// TIA Portal V20 export
FUNCTION_BLOCK "LER_BrakeTest"   // FB103, LAD
// stored: Access Published, MemoryReserve 100, SetENOAutomatically false
   VAR_INPUT
      unitStatus : "LAF_typeUnitStatus";   // Status of the unit
      EnableManualCmds : Bool;
      mcRun : Bool;
      allFDoorClose : Bool;
      allFDoorRelease : Bool;
      allBrakeTestStart : Bool;
      hardwareId : HW_IO;
   END_VAR
   VAR_IN_OUT
      moduleInterface : Bool;
   END_VAR
BEGIN
END_FUNCTION_BLOCK
